TYPE ST_DIS_Inputs :
STRUCT
	bInputCh1 : BOOL;
	bInputCh2 : BOOL;
	bInputCh3 : BOOL;
	bInputCh4 : BOOL;
	bInputCh5 : BOOL;
	bInputCh6 : BOOL;
	bInputCh7 : BOOL;
	bInputCh8 : BOOL;
END_STRUCT
END_TYPE

(* stored: Version 1.1.0.1
   DUT ST_DIS_Inputs: Id {6a40389f-fe8f-407e-bba0-cf326bbc679c} *)
